FUNCTION_BLOCK E_SREN (* Event-driven bistable *)
  (* Standard: 61499-1 Annex A; Description: Copyright (c) 2024 HR Agrartechnik GmbH This program and the accompanying materials are made available under the terms of the Eclipse Public License 2.0 which is available at https://www.eclipse.org/legal/epl-2.0/ SPDX-License-Identifier: EPL-2.0 The Output Q will be TRUE only at S. The Output Q will be FALSE only at R and ERR. The Output Q will be not changed at NONE *)
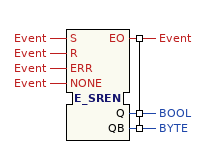
  EVENT_INPUT
    S; (* Enabled (on, active, etc.) *)
    R; (* Disabled (off, passive, etc.) *)
    ERR; (* Error indicator *)
    NONE; (* Not available or not installed *)
  END_EVENT
  EVENT_OUTPUT
    EO WITH Q, QB; (* Output Q has changed *)
  END_EVENT
  VAR_OUTPUT
    Q : BOOL; (* BOOL Output *)
    QB : BYTE := COMMAND_DISABLE; (* 2bit (quarter Byte) Output with 4 States *)
  END_VAR
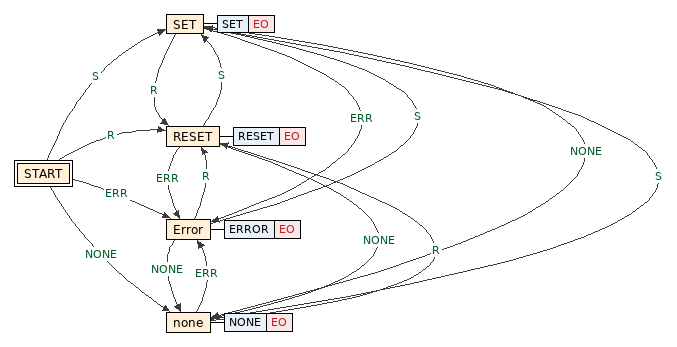
  EC_STATES
    START; (* Initial State *)
    SET : SET -> EO;
    RESET : RESET -> EO;
    Error : ERROR -> EO;
    none : NONE -> EO;
  END_STATES
  EC_TRANSITIONS
    START TO SET := S;
    SET TO RESET := R;
    RESET TO SET := S;
    START TO RESET := R;
    START TO Error := ERR;
    START TO none := NONE;
    RESET TO Error := ERR;
    Error TO RESET := R;
    Error TO none := NONE;
    none TO Error := ERR;
    SET TO Error := ERR;
    RESET TO none := NONE;
    Error TO SET := S;
    none TO RESET := R;
    SET TO none := NONE;
    none TO SET := S;
  END_TRANSITIONS
  ALGORITHM SET IN ST:
Q := TRUE;
QB := COMMAND_ENABLE;
  END_ALGORITHM
  ALGORITHM RESET IN ST:
Q := FALSE;
QB := COMMAND_DISABLE;
  END_ALGORITHM
  ALGORITHM ERROR IN ST:
Q := FALSE;
QB := STATUS_ERROR;
  END_ALGORITHM
  ALGORITHM NONE IN ST:
// Q Don't care/take no action (leave function as is)
QB := COMMAND_NO_ACTION;
  END_ALGORITHM
END_FUNCTION_BLOCK
